TYPE "Motor2Sts"
VERSION : 0.1
// Block: Motor2Sts
   STRUCT
      AlarmPresence : Bool;
      RunBkwPermitted : Bool;
      RunFwdPermitted : Bool;
      Running : Bool;
   END_STRUCT;

END_TYPE
